FUNCTION_BLOCK RepairProducer
  (* Standard: 61499-2 *)
  (* Version 1.0, 2026-07-21, Dimitrios Kalligaridis *)
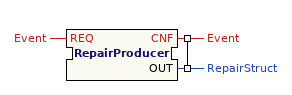
  EVENT_INPUT
    REQ;
  END_EVENT
  EVENT_OUTPUT
    CNF WITH OUT;
  END_EVENT
  VAR_OUTPUT
    OUT : mypackage::RepairStruct;
  END_VAR
END_FUNCTION_BLOCK
